(* CoDeSys 2.3 export: TIME_TO_MMSS.EXP *)

(* POU FUNv1/TIME_TO_MMSS, ST *)
FUNCTION TIME_TO_MMSS : STRING
VAR_INPUT
    t:       TIME;
END_VAR
VAR
    minuta:  DWORD;
    secunda: DWORD;
END_VAR
TIME_TO_MMSS := ':';
minuta       := TIME_TO_DWORD(t) / 60000;
secunda      := TIME_TO_DWORD(t) / 1000 MOD 60;
TIME_TO_MMSS := INSERT(TIME_TO_MMSS, DWORD_TO_STRING(minuta), 0);
IF minuta < 100 THEN
    TIME_TO_MMSS := CONCAT(' ', TIME_TO_MMSS);
END_IF
IF minuta < 10 THEN
    TIME_TO_MMSS := CONCAT(' ', TIME_TO_MMSS);
END_IF
IF secunda < 10 THEN
    TIME_TO_MMSS := CONCAT(TIME_TO_MMSS, '0');
END_IF;
TIME_TO_MMSS := CONCAT(TIME_TO_MMSS, DWORD_TO_STRING(secunda));
END_FUNCTION
